Staubli VAL3: start.pgx

program start()
begin

  // read file
  call util:readFile("Disk://input_day6.txt", sInput)
  // sInput[0] = "1,1,3,5,3,1,....."

  call str:splitString(sInput,",", lResult)

  call util:vec2num(lResult.sString, nInput)
  call util:vec2num(lResult[1].sString, nInput2)

  call util:mergeVectors(nInput,nInput2, nResult)
  call util:vec2num(lResult[2].sString, nInput2)
  call util:mergeVectors(nResult,nInput2, nInput)

  // PUZZLE 1
  call generation_generator(80)
  // 361169

  // PUZZLE 2
  call generation_generator(256)
  // 1634946868992

end
